FUNCTION_BLOCK GF_Entleeren	EXTENDS FB_Basis
VAR_INPUT
	// Instanzieren von Sensoren mit Interfaces
	I_Level			:I_Sensor;
	// Instanzieren von Aktoren mit Interfaces
	I_Ventil		:I_Magnetventil;
	// Rezeptparameter durch Controlword
	I_CW			:RezeptControlWord;
	I_SekReady		:BOOL;
	I_SekActiv		:BOOL;	
END_VAR
VAR_OUTPUT
	O_SW		:RezeptStatusWord;
END_VAR
VAR
	
END_VAR

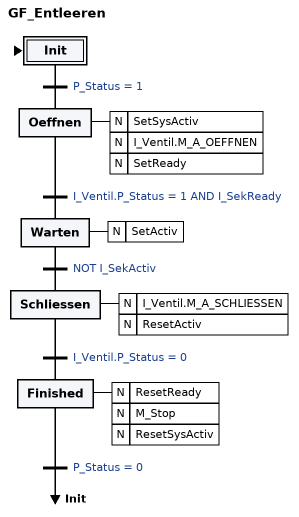
INITIAL_STEP Init:
END_STEP
TRANSITION FROM Init TO Oeffnen
    := P_Status = 1;
END_TRANSITION
STEP Oeffnen:
    SetSysActiv(N);
    I_Ventil.M_A_OEFFNEN(N);
    SetReady(N);
END_STEP
TRANSITION FROM Oeffnen TO Warten
    := I_Ventil.P_Status = 1 AND I_SekReady;
END_TRANSITION
STEP Warten:
    SetActiv(N);
END_STEP
TRANSITION FROM Warten TO Schliessen
    := NOT I_SekActiv;
END_TRANSITION
STEP Schliessen:
    I_Ventil.M_A_SCHLIESSEN(N);
    ResetActiv(N);
END_STEP
TRANSITION FROM Schliessen TO Finished
    := I_Ventil.P_Status = 0;
END_TRANSITION
STEP Finished:
    ResetReady(N);
    M_Stop(N);
    ResetSysActiv(N);
END_STEP
TRANSITION FROM Finished TO Init
    := P_Status = 0;
END_TRANSITION

ACTION ResetActiv:
O_SW.ReactActiv := FALSE;
O_SW.GF2Activ := FALSE;
END_ACTION

ACTION ResetReady:
O_SW.ReactReady := FALSE;
END_ACTION

ACTION ResetSysActiv:
GVL.SysState := 0;
END_ACTION

ACTION SetActiv:
O_SW.ReactActiv := TRUE;
O_SW.GF2Activ := TRUE;
END_ACTION

ACTION SetReady:
O_SW.ReactReady:= TRUE;
END_ACTION

ACTION SetSysActiv:
GVL.SysState := 1;
END_ACTION

END_FUNCTION_BLOCK

(* stored: Version 1.1.0.1, ProductVersion 3.1.4024.12
   POU GF_Entleeren: Id {c2b92295-fb26-4f0a-8170-9b037e32b2ff}, SpecialFunc None
   Folder 01_Aktionen: Id {f5821c1c-9dc8-40f3-a0d4-9b6f5127f676}
   Action ResetActiv: Id {42c1f1d2-5940-49d5-a493-4a56b3ea7031}
   Action ResetReady: Id {992be6a1-03cc-4957-a86e-9e68d4f49100}
   Action ResetSysActiv: Id {32f4ec17-ac4b-4eb9-92bb-7a0d41909dbb}
   Action SetActiv: Id {7eaec211-ab56-45a6-a5cc-30266950cb43}
   Action SetReady: Id {361f3e35-a7a4-4bc9-ba7a-1853d422559d}
   Action SetSysActiv: Id {8b821075-6656-4260-9cda-75120b7a64c9} *)
